% RSLogix 500 project heater_analog.RSS, saved by version 8.30.00.16 %
PROJECT "UNTITLED"    % processor: Bul.1763 MicroLogix 1100 Series B %

PROGRAM FILES
  LAD 2 "MAIN"  4 rungs

DATA FILES
  O0 OUTPUT  8 elements
  I1 INPUT  16 elements
  S2 STATUS  66 elements
  B3 BINARY  1 elements
  T4 TIMER  1 elements
  C5 COUNTER  1 elements
  R6 CONTROL  1 elements
  N7 INTEGER  2 elements
  F8 FLOAT  1 elements
  PD9 TEMP  1 elements

LADDER 2 "MAIN"
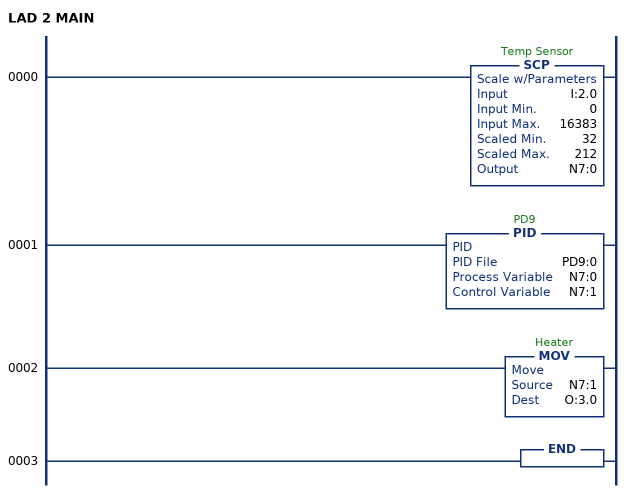
% Rung: 0 %
SOR SCP I:2.0 0 16383 32 212 N7:0 EOR
%   I:2.0  "Temp Sensor Input" %
%   N7:0  "Temp Sensor" %
% Rung: 1 %
SOR PID PD9:0 N7:0 N7:1 EOR
%   PD9:0  PD9 %
%   N7:0  "Temp Sensor" %
%   N7:1  "PID Output" %
% Rung: 2 %
SOR MOV N7:1 O:3.0 EOR
%   N7:1  "PID Output" %
%   O:3.0  "Heater" %
% Rung: 3 %
SOR END EOR

OTHER DOCUMENTED ADDRESSES
  N7:1/0  "Temp Controller"
  O:3.0/0  "Output"
